FUNCTION_BLOCK FB_AtPositionState_Test EXTENDS TcUnit.FB_TestSuite
VAR
    Expected: BOOL;
    Actual: BOOL;
END_VAR

TEST('FB_AtPositionState_Test Dummy Test');
AssertEquals(Expected := Expected,
             Actual := Actual,
             Message := 'Error Message');
TEST_FINISHED();

END_FUNCTION_BLOCK

(* stored: Version 1.1.0.1, ProductVersion 3.1.4022.18
   POU FB_AtPositionState_Test: Id {bf2e9af8-32e4-4631-81c6-8aaefd3f824d}, SpecialFunc None *)
